FUNCTION F_PartIsPresent : BOOL
VAR_INPUT
	WX : sBogie;
END_VAR
VAR
END_VAR

IF WX.A.bPP1_Input AND WX.A.bPP2_Input AND WX.B.bPP1_Input AND WX.A.bPP2_Input THEN
	F_PartIsPresent := 1;
	ELSE
		F_PartIsPresent := 0;
END_IF

END_FUNCTION

(* stored: Version 1.1.0.1, ProductVersion 3.1.4024.12
   POU F_PartIsPresent: Id {4ae60c69-55ae-4f4e-8d5c-b51adb5bfc7c}, SpecialFunc None *)
